FUNCTION_BLOCK FB_List IMPLEMENTS I_List
VAR
    fbMemMan:       FB_DynMem_Manager;
    fbBuffer:       FB_DynMem_Buffer(ipMemMan := fbMemMan);
END_VAR

METHOD AddItem : DINT
VAR_INPUT
    ipObject:       I_Object;
END_VAR
IF ipObject = 0 THEN
    AddItem := -1;
    RETURN;
END_IF

IF THIS^.nCount >= TO_UDINT(GVL_IntegerTypeBounds.DINT_UPPER_BOUND) THEN
    AddItem := -1;
    RETURN;
END_IF

AddItem := THIS^.AppendToBuffer(ipObject);
END_METHOD

METHOD PRIVATE AppendToBuffer : DINT
VAR_INPUT
    ipObject:   I_Object;
END_VAR
VAR
    pTmp:       POINTER TO I_Object;
END_VAR
IF ipObject = 0 THEN
    AppendToBuffer := -1;
    RETURN;
END_IF

THIS^.fbBuffer.Resize(nSize := THIS^.fbBuffer.nBufferSize + SIZEOF(POINTER TO I_Object),
                      bPreserve := TRUE,
                      bReset := FALSE);

pTmp := THIS^.pBuffer;
IF pTmp <> 0 THEN
    pTmp[THIS^.nLastIdx] := ipObject;
END_IF

AppendToBuffer := THIS^.nLastIdx;
END_METHOD

{warning 'add property implementation'}
PROPERTY bIsReadOnly : BOOL
GET
END_GET
END_PROPERTY

METHOD Clear
THIS^.fbBuffer.Resize(nSize := 0,
                      bPreserve := FALSE,
                      bReset := TRUE);
END_METHOD

METHOD Contains : BOOL
VAR_INPUT
    ipObject:       I_Object;
END_VAR
VAR
    i:              DINT;
    ipTmp:          I_Object;
END_VAR
IF ipObject = 0 THEN
    RETURN;
END_IF

FOR i := 0 TO THIS^.nLastIdx DO
    IF F_CompareObjects(ipObject, THIS^.ItemAt(i)) THEN
        Contains := TRUE;
        RETURN;
    END_IF
END_FOR
END_METHOD

{warning 'add method implementation '}
METHOD CopyFrom
VAR_INPUT
END_VAR
END_METHOD

METHOD FB_init : BOOL
VAR_INPUT
	bInitRetains : BOOL; // if TRUE, the retain variables are initialized (warm start / cold start)
	bInCopyCode : BOOL;  // if TRUE, the instance afterwards gets moved into the copy code (online change)
END_VAR
THIS^.fbBuffer.CreateBuffer(nSize := 0, bReset := TRUE);
END_METHOD

METHOD IndexOfItem : DINT
VAR_INPUT
    ipObject:   I_Object;
END_VAR
VAR
    i:          DINT;
END_VAR
IF ipObject = 0 THEN
    IndexOfItem := -1;
    RETURN;
END_IF

FOR i := 0 TO THIS^.nLastIdx DO
    IF F_CompareObjects(THIS^.ItemAt(i), ipObject) THEN
        IndexOfItem := i;
        RETURN;
    END_IF
END_FOR

IndexOfItem := -1;
END_METHOD

{warning 'add method implementation '}
METHOD Insert : BOOL
VAR_INPUT
	(* Zero-based index at which object should be inserted*)
	nIdx	: DINT;
	(* Object to be inserted*)
	ipObject	: I_Object;
END_VAR
END_METHOD

METHOD ItemAt : I_Object
VAR_INPUT
    nIdx:       DINT;
END_VAR
VAR
    pTmp:       POINTER TO I_Object;
END_VAR
pTmp := THIS^.fbBuffer.pBuffer;
IF nIdx >= 0
    AND_THEN nIdx <= GVL_IntegerTypeBounds.DINT_UPPER_BOUND
    AND_THEN pTmp <> 0 THEN
    ItemAt := pTmp[nIdx];
END_IF
END_METHOD

{warning 'add method implementation '}
METHOD LastIndexOf : DINT
VAR_INPUT
END_VAR
END_METHOD

{warning 'add property implementation'}
PROPERTY nCount : UDINT
GET
IF THIS^.fbBuffer.nBufferSize > 0 THEN
    nCount := TO_UDINT(THIS^.nLastIdx) + 1;
ELSE
    nCount := 0;
END_IF
END_GET
END_PROPERTY

PROPERTY PRIVATE nLastIdx : DINT
GET
IF THIS^.fbBuffer.nBufferSize > 0 THEN
    nLastIdx := TO_DINT(THIS^.fbBuffer.nBufferSize/SIZEOF(POINTER TO I_Object) - 1);
ELSE
    nLastIdx := 0;
END_IF
END_GET
END_PROPERTY

PROPERTY PROTECTED pBuffer : POINTER TO I_Object
GET
pBuffer := THIS^.fbBuffer.pBuffer;
END_GET
END_PROPERTY

{warning 'add method implementation '}
METHOD Remove : BOOL
VAR_INPUT
    ipObject:   I_Object;
END_VAR
VAR
    i:          DINT;
END_VAR
IF ipObject = 0 THEN
    RETURN;
END_IF
END_METHOD

METHOD RemoveAt : BOOL
VAR_INPUT
    nIdx:       DINT;
END_VAR
VAR
    pBuffer:    POINTER TO I_Object;
    pTmp:       POINTER TO BYTE;
    nTmpLength: UDINT;
END_VAR
IF NOT THIS^.ValidateIndex(nIdx) THEN
    RETURN;
END_IF

nTmpLength := THIS^.fbBuffer.nBufferSize - SIZEOF(POINTER TO I_Object);
pTmp := __NEW(BYTE, nTmpLength);

pBuffer := THIS^.pBuffer;
Tc2_System.MEMCPY(destAddr := pTmp,
                  srcAddr := pBuffer,
                  n := TO_UDINT(nIdx));

IF nIdx < THIS^.nLastIdx THEN
    Tc2_System.MEMCPY(destAddr := pTmp,
                      srcAddr := ADR(pBuffer[nIdx + 1]),
                      n := TO_UDINT(THIS^.nLastIdx - nIdx));
END_IF

THIS^.fbBuffer.Resize(nSize := nTmpLength,
                      bPreserve := FALSE,
                      bReset := TRUE);

Tc2_System.MEMCPY(destAddr := THIS^.pBuffer,
                  srcAddr := pTmp,
                  n := nTmpLength);

IF pTmp <> 0 THEN
    __DELETE(pTmp);
END_IF

RemoveAt := TRUE;
END_METHOD

METHOD PRIVATE ValidateIndex : BOOL
VAR_INPUT
    nIdx:       DINT;
END_VAR
ValidateIndex := (0 <= nIdx) AND_THEN (nIdx <= THIS^.nLastIdx);
END_METHOD

END_FUNCTION_BLOCK

(* stored: Version 1.1.0.1, ProductVersion 3.1.4024.12
   POU FB_List: Id {3d09efba-b29b-0efb-0296-650e9b624057}, SpecialFunc None
   Method AddItem: Id {6b056280-a8e0-0e09-074f-1d3cb2b9d2ee}
   Method AppendToBuffer: Id {94a09fe7-a3b1-0757-3845-78a783dfa8df}
   Property bIsReadOnly: Id {ea05ed59-e6d5-04a8-1de2-ffb7506213f8}
   Get Get: Id {a4d9e74a-16d7-0e1b-1c5e-f81bb0e3b24c}
   Method Clear: Id {a137cbbb-95f2-09f4-3dc3-74fa015dc829}
   Method Contains: Id {e8902ae8-937d-0e9c-2799-5637622ee1a4}
   Method CopyFrom: Id {82fd7cfd-ccea-4821-9028-f218afcf0f77}
   Method FB_init: Id {8965c983-9c90-0eff-34d5-5f9bc7e316ec}
   Method IndexOfItem: Id {f7e53ae0-cf34-07c7-1000-7e57010e6b64}
   Method Insert: Id {77a6d124-8e25-0160-2603-5cc7fd52e20d}
   Method ItemAt: Id {238f3b9c-2aef-0eae-1903-43fa04efd7f9}
   Method LastIndexOf: Id {8e4f2e47-21f3-40ec-b58f-1dd566a9f877}
   Property nCount: Id {1f12488a-7040-079f-323b-3cb46e3d0c32}
   Get Get: Id {bb42c317-8361-0ccf-0e90-3eba5d86d3f8}
   Property nLastIdx: Id {f5b11e21-f8ae-0e25-3022-1dce5f47fd43}
   Get Get: Id {1cd81378-769b-0500-1fca-8e5a97da3e08}
   Property pBuffer: Id {77e9ccb7-bd64-0330-2eb7-1b02a4db0799}
   Get Get: Id {33c39764-3862-0df0-0390-31060a2252c6}
   Method Remove: Id {c78f7a59-fd40-0868-172c-5551d6ad8aa7}
   Method RemoveAt: Id {815f2227-6866-0206-0e82-6f52e1ffa7b5}
   Method ValidateIndex: Id {0ea38052-127a-471c-bdf2-c6656fc2dff6} *)
